// TIA Portal V18 export
// export: Created 2026-01-09T11:31:56.254394Z, ExportSetting WithDefaults, DisplayName Totally Integrated Automation Portal, DisplayVersion V18 Update 5, DisplayName TIA Portal Openness, DisplayVersion V18 Update 5, DisplayName TIA Portal Teamcenter Gateway, DisplayVersion V18, DisplayName TIA Portal Version Control Interface, DisplayVersion V18, DisplayName SINAMICS Startdrive Advanced, DisplayVersion V18 SP2 Update 1, DisplayName SINAMICS Startdrive G110M, G120, G120C, G120D, G120P, G115D, DisplayVersion V18 SP2 Update 1, DisplayName SINAMICS Startdrive G130, G150, S120, S150, SINAMICS MV, S210, G220, S200, DisplayVersion V18 SP2 Update 1, DisplayName STEP 7 Professional, DisplayVersion V18 Update 5, DisplayName STEP 7 Safety, DisplayVersion V18, DisplayName WinCC Professional, DisplayVersion V18 Update 5
TagTable "Robot"
  Robot_DB_Control_Robot1GripControl : Bool  (PLC tag Robot_DB.Control.Robot1GripControl, CPU S71500-2PN_TP700, 1 s)
  Robot_DB_Control_Robot2GripControl : Bool  (PLC tag Robot_DB.Control.Robot2GripControl, CPU S71500-2PN_TP700, 1 s)
  Robot_DB_Control_Robot3GripControl : Bool  (PLC tag Robot_DB.Control.Robot3GripControl, CPU S71500-2PN_TP700, 1 s)
  KukaRobot1_CtrlDB_sHMI : KukaRobot_HMI  (PLC tag KukaRobot1_CtrlDB.sHMI, CPU S71500-2PN_TP700, 1 s)
    TagStructureMember "PGNO_PBIT"
    TagStructureMember "EXT_START"
    TagStructureMember "MOVE_ENABLE"
    TagStructureMember "CONF_MESS"
    TagStructureMember "DRIVES_OFF"
    TagStructureMember "DRIVES_ON"
    TagStructureMember "I_O_ACT"
    TagStructureMember "RC_RDY1"
    TagStructureMember "ALARM_STOP"
    TagStructureMember "USER_SAF"
    TagStructureMember "PERI_RDY"
    TagStructureMember "ROB_CAL"
    TagStructureMember "I_O_ACTCONF"
    TagStructureMember "STOPMESS"
    TagStructureMember "ALARM_STOP_INTERN"
    TagStructureMember "PGNO_FBIT_REFL"
    TagStructureMember "PRO_ACT"
    TagStructureMember "APPL_RUN"
    TagStructureMember "PRO_MOVE"
    TagStructureMember "IN_HOME"
    TagStructureMember "ON_PATH"
    TagStructureMember "NEAR_POSRET"
    TagStructureMember "T1"
    TagStructureMember "T2"
    TagStructureMember "AUT"
    TagStructureMember "EXT"
    TagStructureMember "TaskMode"
    TagStructureMember "PartType"
    TagStructureMember "SpeedSet"
    TagStructureMember "HomeSeqStart"
    TagStructureMember "AutoCycleStart"
    TagStructureMember "CurrentMode"
    TagStructureMember "CurrentPartType"
    TagStructureMember "SpeedActual"
    TagStructureMember "ProgramSequence"
    TagStructureMember "WaitForHomeSeqStart"
    TagStructureMember "GoHomeFail"
    TagStructureMember "HomeSeqOK"
    TagStructureMember "WaitForAutoCycleStart"
    TagStructureMember "iTaskMode"
    TagStructureMember "iPartType"
    TagStructureMember "iSpeedValue"
    TagStructureMember "iPGNO"
    TagStructureMember "AutoStart"
    TagStructureMember "SrartHome"
    TagStructureMember "StartAutoCycle"
    TagStructureMember "Ready"
    TagStructureMember "StartComplete"
    TagStructureMember "StartUpTimeOut"
    TagStructureMember "Warning"
    TagStructureMember "Error"
    TagStructureMember "ErrorCode"
    TagStructureMember "Seconds"
    TagStructureMember "Minute"
    TagStructureMember "Hours"
    TagStructureMember "CountPulse"
    TagStructureMember "StartSeq"
  KukaRobot2_CtrlDB_sHMI : KukaRobot_HMI  (PLC tag KukaRobot2_CtrlDB.sHMI, CPU S71500-2PN_TP700, 1 s)
    TagStructureMember "PGNO_PBIT"
    TagStructureMember "EXT_START"
    TagStructureMember "MOVE_ENABLE"
    TagStructureMember "CONF_MESS"
    TagStructureMember "DRIVES_OFF"
    TagStructureMember "DRIVES_ON"
    TagStructureMember "I_O_ACT"
    TagStructureMember "RC_RDY1"
    TagStructureMember "ALARM_STOP"
    TagStructureMember "USER_SAF"
    TagStructureMember "PERI_RDY"
    TagStructureMember "ROB_CAL"
    TagStructureMember "I_O_ACTCONF"
    TagStructureMember "STOPMESS"
    TagStructureMember "ALARM_STOP_INTERN"
    TagStructureMember "PGNO_FBIT_REFL"
    TagStructureMember "PRO_ACT"
    TagStructureMember "APPL_RUN"
    TagStructureMember "PRO_MOVE"
    TagStructureMember "IN_HOME"
    TagStructureMember "ON_PATH"
    TagStructureMember "NEAR_POSRET"
    TagStructureMember "T1"
    TagStructureMember "T2"
    TagStructureMember "AUT"
    TagStructureMember "EXT"
    TagStructureMember "TaskMode"
    TagStructureMember "PartType"
    TagStructureMember "SpeedSet"
    TagStructureMember "HomeSeqStart"
    TagStructureMember "AutoCycleStart"
    TagStructureMember "CurrentMode"
    TagStructureMember "CurrentPartType"
    TagStructureMember "SpeedActual"
    TagStructureMember "ProgramSequence"
    TagStructureMember "WaitForHomeSeqStart"
    TagStructureMember "GoHomeFail"
    TagStructureMember "HomeSeqOK"
    TagStructureMember "WaitForAutoCycleStart"
    TagStructureMember "iTaskMode"
    TagStructureMember "iPartType"
    TagStructureMember "iSpeedValue"
    TagStructureMember "iPGNO"
    TagStructureMember "AutoStart"
    TagStructureMember "SrartHome"
    TagStructureMember "StartAutoCycle"
    TagStructureMember "Ready"
    TagStructureMember "StartComplete"
    TagStructureMember "StartUpTimeOut"
    TagStructureMember "Warning"
    TagStructureMember "Error"
    TagStructureMember "ErrorCode"
    TagStructureMember "Seconds"
    TagStructureMember "Minute"
    TagStructureMember "Hours"
    TagStructureMember "CountPulse"
    TagStructureMember "StartSeq"
  KukaRobot3_CtrlDB_sHMI : KukaRobot_HMI  (PLC tag KukaRobot3_CtrlDB.sHMI, CPU S71500-2PN_TP700, 1 s)
    TagStructureMember "PGNO_PBIT"
    TagStructureMember "EXT_START"
    TagStructureMember "MOVE_ENABLE"
    TagStructureMember "CONF_MESS"
    TagStructureMember "DRIVES_OFF"
    TagStructureMember "DRIVES_ON"
    TagStructureMember "I_O_ACT"
    TagStructureMember "RC_RDY1"
    TagStructureMember "ALARM_STOP"
    TagStructureMember "USER_SAF"
    TagStructureMember "PERI_RDY"
    TagStructureMember "ROB_CAL"
    TagStructureMember "I_O_ACTCONF"
    TagStructureMember "STOPMESS"
    TagStructureMember "ALARM_STOP_INTERN"
    TagStructureMember "PGNO_FBIT_REFL"
    TagStructureMember "PRO_ACT"
    TagStructureMember "APPL_RUN"
    TagStructureMember "PRO_MOVE"
    TagStructureMember "IN_HOME"
    TagStructureMember "ON_PATH"
    TagStructureMember "NEAR_POSRET"
    TagStructureMember "T1"
    TagStructureMember "T2"
    TagStructureMember "AUT"
    TagStructureMember "EXT"
    TagStructureMember "TaskMode"
    TagStructureMember "PartType"
    TagStructureMember "SpeedSet"
    TagStructureMember "HomeSeqStart"
    TagStructureMember "AutoCycleStart"
    TagStructureMember "CurrentMode"
    TagStructureMember "CurrentPartType"
    TagStructureMember "SpeedActual"
    TagStructureMember "ProgramSequence"
    TagStructureMember "WaitForHomeSeqStart"
    TagStructureMember "GoHomeFail"
    TagStructureMember "HomeSeqOK"
    TagStructureMember "WaitForAutoCycleStart"
    TagStructureMember "iTaskMode"
    TagStructureMember "iPartType"
    TagStructureMember "iSpeedValue"
    TagStructureMember "iPGNO"
    TagStructureMember "AutoStart"
    TagStructureMember "SrartHome"
    TagStructureMember "StartAutoCycle"
    TagStructureMember "Ready"
    TagStructureMember "StartComplete"
    TagStructureMember "StartUpTimeOut"
    TagStructureMember "Warning"
    TagStructureMember "Error"
    TagStructureMember "ErrorCode"
    TagStructureMember "Seconds"
    TagStructureMember "Minute"
    TagStructureMember "Hours"
    TagStructureMember "CountPulse"
    TagStructureMember "StartSeq"
  KukaRobot1_PalletCount_1 : Int  (PLC tag Robot_DB.Robot_1.PalletCount_1, CPU S71500-2PN_TP700, 100 ms)
  KukaRobot2_PalletCount_1 : Int  (PLC tag Robot_DB.Robot_2.PalletCount_1, CPU S71500-2PN_TP700, 100 ms)
  KukaRobot2_PalletCount_2 : Int  (PLC tag Robot_DB.Robot_2.PalletCount_2, CPU S71500-2PN_TP700, 100 ms)
  KukaRobot3_PalletCount_1 : Int  (PLC tag Robot_DB.Robot_3.PalletCount_1, CPU S71500-2PN_TP700, 100 ms)
  KukaRobot3_PalletCount_2 : Int  (PLC tag Robot_DB.Robot_3.PalletCount_2, CPU S71500-2PN_TP700, 100 ms)
  KukaRobot1_CtrlDB_iSpeedValue : USInt  (PLC tag KukaRobot1_CtrlDB.iSpeedValue, CPU S71500-2PN_TP700, 100 ms)
  KukaRobot2_CtrlDB_iSpeedValue : USInt  (PLC tag KukaRobot2_CtrlDB.iSpeedValue, CPU S71500-2PN_TP700, 100 ms)
  KukaRobot3_CtrlDB_iSpeedValue : USInt  (PLC tag KukaRobot3_CtrlDB.iSpeedValue, CPU S71500-2PN_TP700, 100 ms)
  AutoProcessControl_Robot_3_PalletFull : Bool  (PLC tag AutoProcessControl.Robot_3.PalletFull, CPU S71500-2PN_TP700, 1 s)
  AutoProcessControl_Robot_1_ClearPart : Bool  (PLC tag AutoProcessControl.Robot_1.ClearPart, CPU S71500-2PN_TP700, 1 s)
  ChangeOver_DB_Robot_1_HMI_MaintenancePosReqSel : Bool  (PLC tag ChangeOver_DB.Robot_1.HMI_MaintenancePosReqSel, CPU S71500-2PN_TP700, 1 s)
  ChangeOver_DB_Robot_1_HMI_MaintenancePosActive : Bool  (PLC tag ChangeOver_DB.Robot_1.HMI_MaintenancePosActive, CPU S71500-2PN_TP700, 1 s)
  ChangeOver_DB_Robot_1_HMI_MaintenanceHomeReq : Bool  (PLC tag ChangeOver_DB.Robot_1.HMI_MaintenanceHomeReq, CPU S71500-2PN_TP700, 1 s)
  ChangeOver_DB_Robot_1_MaintenancePosReqSelFlag : Bool  (PLC tag ChangeOver_DB.Robot_1.MaintenancePosReqSelFlag, CPU S71500-2PN_TP700, 1 s)
  ChangeOver_DB_Robot_2_HMI_MaintenancePosReqSel : Bool  (PLC tag ChangeOver_DB.Robot_2.HMI_MaintenancePosReqSel, CPU S71500-2PN_TP700, 1 s)
  ChangeOver_DB_Robot_2_HMI_MaintenancePosActive : Bool  (PLC tag ChangeOver_DB.Robot_2.HMI_MaintenancePosActive, CPU S71500-2PN_TP700, 1 s)
  ChangeOver_DB_Robot_2_HMI_MaintenanceHomeReq : Bool  (PLC tag ChangeOver_DB.Robot_2.HMI_MaintenanceHomeReq, CPU S71500-2PN_TP700, 1 s)
  ChangeOver_DB_Robot_2_MaintenancePosReqSelFlag : Bool  (PLC tag ChangeOver_DB.Robot_2.MaintenancePosReqSelFlag, CPU S71500-2PN_TP700, 1 s)
  ChangeOver_DB_Robot_3_HMI_MaintenancePosReqSel : Bool  (PLC tag ChangeOver_DB.Robot_3.HMI_MaintenancePosReqSel, CPU S71500-2PN_TP700, 1 s)
  ChangeOver_DB_Robot_3_HMI_MaintenancePosActive : Bool  (PLC tag ChangeOver_DB.Robot_3.HMI_MaintenancePosActive, CPU S71500-2PN_TP700, 1 s)
  ChangeOver_DB_Robot_3_HMI_MaintenanceHomeReq : Bool  (PLC tag ChangeOver_DB.Robot_3.HMI_MaintenanceHomeReq, CPU S71500-2PN_TP700, 1 s)
  ChangeOver_DB_Robot_3_MaintenancePosReqSelFlag : Bool  (PLC tag ChangeOver_DB.Robot_3.MaintenancePosReqSelFlag, CPU S71500-2PN_TP700, 1 s)
  Robot3HomeRunning : Bool  (PLC tag KukaRobot3_CtrlDB.sROBtoPLC.User.Cycle.DO300_HomeInside, CPU S71500-2PN_TP700, 1 s)
  Robot1HomeRunning : Bool  (PLC tag KukaRobot1_CtrlDB.sROBtoPLC.User.Cycle.DO300_HomeInside, CPU S71500-2PN_TP700, 1 s)
  Robot2HomeRunning : Bool  (PLC tag KukaRobot2_CtrlDB.sROBtoPLC.User.Cycle.DO300_HomeInside, CPU S71500-2PN_TP700, 1 s)
  ST10_RecipeDB_ParameterElement_Robot1_Ring1Weight : Int  (PLC tag ChangeOver_DB.Robot1.Ring1Weight, CPU S71500-2PN_TP700, 1 s)
  ST10_RecipeDB_ParameterElement_Robot1_ShaftWeight : Int  (PLC tag ChangeOver_DB.Robot1.ShaftWeight, CPU S71500-2PN_TP700, 1 s)
  ST10_RecipeDB_ParameterElement_Robot1_MagnetWeight : Int  (PLC tag ChangeOver_DB.Robot1.MagnetWeight, CPU S71500-2PN_TP700, 1 s)
  ST10_RecipeDB_ParameterElement_Robot1_Ring2Weight : Int  (PLC tag ChangeOver_DB.Robot1.Ring2Weight, CPU S71500-2PN_TP700, 1 s)
  ST10_RecipeDB_ParameterElement_Robot2_Ring1Weight : Int  (PLC tag ChangeOver_DB.Robot2.Ring1Weight, CPU S71500-2PN_TP700, 1 s)
  ST10_RecipeDB_ParameterElement_Robot2_ShaftWeight : Int  (PLC tag ChangeOver_DB.Robot2.ShaftWeight, CPU S71500-2PN_TP700, 1 s)
  ST10_RecipeDB_ParameterElement_Robot2_MagnetWeight : Int  (PLC tag ChangeOver_DB.Robot2.MagnetWeight, CPU S71500-2PN_TP700, 1 s)
  ST10_RecipeDB_ParameterElement_Robot2_Ring2Weight : Int  (PLC tag ChangeOver_DB.Robot2.Ring2Weight, CPU S71500-2PN_TP700, 1 s)
  ST10_RecipeDB_ParameterElement_Robot3_Ring1Weight : Int  (PLC tag ChangeOver_DB.Robot3.Ring1Weight, CPU S71500-2PN_TP700, 1 s)
  ST10_RecipeDB_ParameterElement_Robot3_ShaftWeight : Int  (PLC tag ChangeOver_DB.Robot3.ShaftWeight, CPU S71500-2PN_TP700, 1 s)
  ST10_RecipeDB_ParameterElement_Robot3_MagnetWeight : Int  (PLC tag ChangeOver_DB.Robot3.MagnetWeight, CPU S71500-2PN_TP700, 1 s)
  ST10_RecipeDB_ParameterElement_Robot3_Ring2Weight : Int  (PLC tag ChangeOver_DB.Robot3.Ring2Weight, CPU S71500-2PN_TP700, 1 s)
  Robot_DB_Robot_1_BrakeTest_Req : Bool  (PLC tag Robot_DB.Robot_1.BrakeTest_Req, CPU S71500-2PN_TP700, 1 s)
  Robot_DB_Robot_2_BrakeTest_Req : Bool  (PLC tag Robot_DB.Robot_2.BrakeTest_Req, CPU S71500-2PN_TP700, 1 s)
  Robot_DB_Robot_3_BrakeTest_Req : Bool  (PLC tag Robot_DB.Robot_3.BrakeTest_Req, CPU S71500-2PN_TP700, 1 s)
